{attribute 'qualified_only'}
VAR_GLOBAL
	// Pitch Mechanism:
	{attribute 'TcLinkTo' := '.diEncCnt:=TIIB[EL5042_M1K2_Pitch]^FB Inputs Channel 1^Position'}
	M1K2_Pitch : HOMS_PitchMechanism := (ReqPosLimHi := 25824,
		                                 ReqPosLimLo := 25680,
		                                 diEncPosLimHi := 10097184,
		                                 diEncPosLimLo := 10040880); // Set to 50 urad before hard limits tripped during SAT
END_VAR

(* stored: Version 1.1.0.1, ProductVersion 3.1.4022.18
   GVL GVL_M1K2: Id {2074b16f-0d4c-4051-96e9-b5e1650ca1c7} *)
